// TIA Portal V20 export
TYPE "LConSMC_typeAxisStartupData"
// stored: Access Published
   STRUCT
      typeOfAxis : Int;
      communicationOK : Bool;
      inOperation : Bool;
      torqueDataEnabled : Bool;
      adaptionState : DInt;
      referenceTorque : LReal;
      loadGear : "LConSMC_typeLoadGear";
      leadScrew : LReal;
      axisLengthUnit : UDInt;   // Length unit of TO (see TO.Units.LengthUnit) !Only necessary if "getAxisConfigAtStart" = FALSE and for Sectional Drives!
      velocityUnit { S7_SetPoint := 'True'} : UDInt;
      torqueUnit : UDInt;
      axisDefaultAcceleration : LReal;
      axisDefaultJerk : LReal;
   END_STRUCT;
END_TYPE
